PROGRAM MAIN
VAR
	fbClock	: FB_Toggle;
	fbTrafficLight_enum	: FB_TrafficLight_ENUM;
	fbTrafficLight_stp	: FB_TrafficLight_STP;
END_VAR

fbClock();
fbTrafficLight_enum();
fbTrafficLight_stp();

END_PROGRAM

(* stored: Version 1.1.0.1, ProductVersion 3.1.4024.12
   POU MAIN: Id {79d0d9a2-6072-47c5-b5c5-45b55f6a637d}, SpecialFunc None *)
